INTERFACE I_AsyncResponseHeaderAccessor

METHOD PUBLIC TryGetResponseIdFromRequest : BOOL
VAR_INPUT
	Request : I_Request;
	Destination : ANY;
END_VAR
END_METHOD

METHOD PUBLIC TryGetSessionIdFromRequest : BOOL
VAR_INPUT
	Request : I_Request;
	Destination : REFERENCE TO T_MAXSTRING;
END_VAR
END_METHOD

METHOD PUBLIC TryGetSessionIdFromResponse : BOOL
VAR_INPUT
	Response : I_ServerResponse;
	Destination : ANY;
END_VAR
END_METHOD

END_INTERFACE

(* stored: Version 1.1.0.1, ProductVersion 3.1.4026.13
   Itf I_AsyncResponseHeaderAccessor: Id {61b9a4ee-8cd0-4644-b0b2-453653811270}
   Method TryGetResponseIdFromRequest: Id {5a578aba-db65-4303-a492-398025f4f169}
   Method TryGetSessionIdFromRequest: Id {59ffb8d0-e7f1-4d58-ade8-d6555afd94d8}
   Method TryGetSessionIdFromResponse: Id {8962ab21-3edc-4974-917e-ae01e1fac701} *)
